{attribute 'conditionalshow'}
TYPE ST_UN_FLOAT_CONVERT_DWORD_REAL :
UNION
	{attribute 'hide'}
	dwRawValue				: DWORD;											//Raw value as dword
	{attribute 'hide'}
	rValueFloat				: REAL;												//Float value
END_UNION
END_TYPE

(* stored: Version 1.1.0.1, ProductVersion 3.1.4024.9
   DUT ST_UN_FLOAT_CONVERT_DWORD_REAL: Id {b586da3b-10f1-422f-b5a9-972164396840} *)
